PROGRAM PRG_CASE_FinaliseDataManual
VAR
	fbCase_FinaliseData		: FB_CASE_FinaliseData;
	
	(* Init function/method declarations*)
	rTrigDataInit		: R_TRIG;
	bDataInit			: BOOL;
	iOuter				: INT;
	iPack				: INT;
	sPackNum			: STRING;
	sOuterNum			: STRING;
	sPackCode			: STRING;
	
	(* Inputs *)
	bExecute 				: BOOL;		(* set TRUE to move Outers *)
	bDoorReject				: BOOL;
	stRejectReasonsForCase	: ST_RejectReasonsForCase; //inicjalizacja rejectResonow
	
	(* In/Out *)
	stProductInstruction	: ST_PCM_Status;
	stCodeInfo_Outer		: ST_CodeInfo;
	stCACData 				: ST_CAC_Data;	(* Case Queue *)
	stCACDataHMI			: ST_HMI_CAC_Data;
	
	(* Outputs *)
	bDone 					: BOOL;
	bBusy					: BOOL;

	bCACValid				: BOOL;
	bCACInvalid				: BOOL;

	bCheckDuplicates		: BOOL;
	bReadyToValidate		: BOOL;
	
	sRejectCode				: T_MaxString;
	sCaseContent			: T_LongSTRING;
	
END_VAR

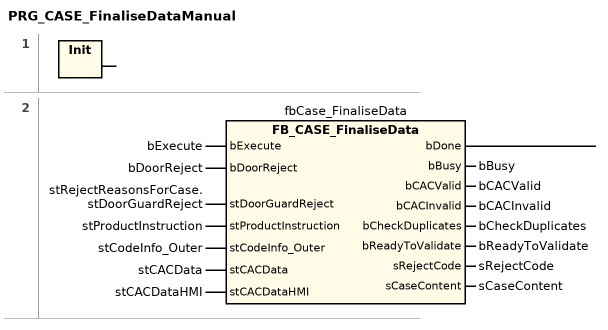
// NETWORK 1
Init();

// NETWORK 2
fbCase_FinaliseData(
    bExecute := bExecute,
    bDoorReject := bDoorReject,
    stDoorGuardReject := stRejectReasonsForCase.stDoorGuardReject,
    stProductInstruction := stProductInstruction,
    stCodeInfo_Outer := stCodeInfo_Outer,
    stCACData := stCACData,
    stCACDataHMI := stCACDataHMI,
    bBusy => bBusy,
    bCACValid => bCACValid,
    bCACInvalid => bCACInvalid,
    bCheckDuplicates => bCheckDuplicates,
    bReadyToValidate => bReadyToValidate,
    sRejectCode => sRejectCode,
    sCaseContent => sCaseContent); // FB_CASE_FinaliseData

ACTION Init:

rTrigDataInit(CLK := bDataInit);

IF rTrigDataInit.Q THEN
	
stProductInstruction.nOutersPerCase		:= 50;
stProductInstruction.nPacksPerOuter 	:= 10;

	FOR iOuter := 1 TO stProductInstruction.nOutersPerCase DO
		(* Ustaw outer *)
		stCACData.Outer[iOuter].Barcode    := CONCAT('OUTER', F_StringAddPrefix(INT_TO_STRING(iOuter),2,'0'));
		stCACData.Outer[iOuter].OuterCodeStatus := 5;
		
		FOR iPack := 1 TO stProductInstruction.nPacksPerOuter DO
			(* Pack number z zerami *)
			sPackNum := CONCAT('0', INT_TO_STRING(iPack));  (* dla 1-9: '01'-'09' *)
			IF iPack = 10 THEN
				sPackNum := '10';
			END_IF;
			
			(* Outer number z zerami dla 1-9 *)
			sOuterNum := CONCAT('0', INT_TO_STRING(iOuter));
			IF iOuter >= 10 THEN
				sOuterNum := INT_TO_STRING(iOuter);
			END_IF;
			
			(* Sklej pack code *)
			sPackCode := CONCAT(CONCAT('PACK', sPackNum), CONCAT('OUTER', sOuterNum));
			
			(* Przypisz *)
			stCACData.Outer[iOuter].PackCode[iPack]			:= sPackCode;
			stCACData.Outer[iOuter].PackCodeStatus[iPack]	:= 5;
			stCACData.Outer[iOuter].PackRejectID[iPack]		:= 0;
			
		END_FOR;
	END_FOR;	
	
END_IF

//initialize needed data structures
stCACData.NumberOfOuters				:= stProductInstruction.nOutersPerCase;
stCodeInfo_Outer.nEntireLength					:= 7;
stCodeInfo_Outer.stSerialCode.nCodeStartPos 	:= 1;
stCodeInfo_Outer.stSerialCode.nCodeLength 		:= 7;
END_ACTION

END_PROGRAM

(* stored: Version 1.1.0.1
   POU PRG_CASE_FinaliseDataManual: Id {de1c4946-2f6a-46af-94e8-69091e414096}, SpecialFunc None
   Action Init: Id {08194a4d-05fa-4272-8ec8-ee3a74e4e1b9} *)
